FUNCTION_BLOCK SampleTaskIteration EXTENDS TcoCore.TcoTask
VAR	
	_x : LREAL;
	_y : LREAL;
	_d : LREAL;
	{attribute addProperty Minimum 100}
	{attribute addProperty Maximum 1000}
	_iterations : INT;	
	_currentIteration : INT;	
END_VAR

IF(Execute()) THEN
	_y := SIN(_x);
	_x := _x + _d;		
	_currentIteration := _currentIteration + 1;	
	DoneWhen(_currentIteration >= _iterations);
END_IF

(*~
	<docu>
		<summary>
			Restores this instance to the Ready state. Can be called explicitly or from within one of the restore mechanisms.
			<para>
				See also <see cref="PlcDocu.TcoCore.TcoTask.AutoRestorable()"/>
			</para>
		</summary>			
	</docu>	
~*)
METHOD Restore : ITcoRestorable
SUPER^.Restore();
_x := 0.0;
_y := 0.0;
_currentIteration := 0;
END_METHOD

END_FUNCTION_BLOCK

(* stored: Version 1.1.0.1, ProductVersion 3.1.4024.9
   POU SampleTaskIteration: Id {d1ab64f5-1332-0075-0062-208284e70814}, SpecialFunc None
   Method Restore: Id {418ca9c4-083f-0907-23e2-93b0ad7066ce} *)
